FUNCTION_BLOCK SS4_ifb_Laser_2 (* Basic FB with empty ECC *)
  (* Standard: 61499-2 *)
  (* Version 1.0, 2025-05-06, DEVIASH *)
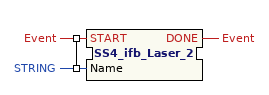
  EVENT_INPUT
    START WITH Name;
  END_EVENT
  EVENT_OUTPUT
    DONE;
  END_EVENT
  VAR_INPUT
    Name : STRING;
  END_VAR
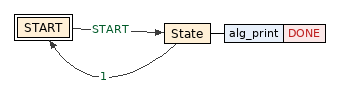
  EC_STATES
    START; (* Initial State *)
    State : alg_print -> DONE;
  END_STATES
  EC_TRANSITIONS
    START TO State := START;
    State TO START := 1;
  END_TRANSITIONS
  ALGORITHM alg_print IN ST:

  END_ALGORITHM
END_FUNCTION_BLOCK
